// Mitsubishi GX Works2 project: k13   PLC: Q02/Q02H

PROGRAM MAIN
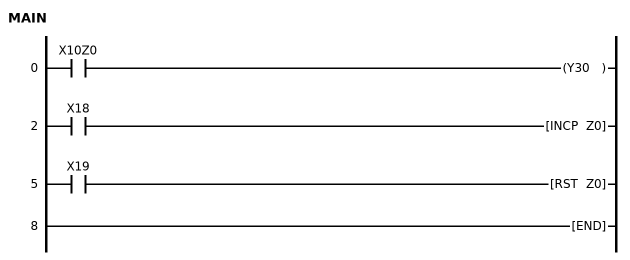
0     LD      X10Z0
      OUT     Y30
2     LD      X18
      INCP    Z0
5     LD      X19
      RST     Z0
8     END
END_PROGRAM
